(* Schneider Machine Expert - Basic project AND Gate, file version 2.9.0.0 *)
(* ProjectInformations: Name=New project *)

HARDWARE
  Cpu 0: TM221C24R
  EthernetConfiguration: NetworkName=M221, IpAllocationMode=FixedAddress, IpAddress=0.0.0.0, SubnetMask=0.0.0.0
  SerialLineConfiguration: Baud=Baud19200, Parity=ParityEven, DataBits=DataBits8, StopBits=StopBits1, PhysicalMedium=PhysicalMediumRs485, SlaveId=1, Addressing=SlaveAddressing
  MastTask: UsePeriodScanMode=false, PeriodScan=100
  FastTask: Period=255
  CpuBehavior: StartingMode=StartAsPreviousState, AutoSaveRamOnEeprom=true, WatchdogPeriod=250

SYMBOLS  (address, symbol, comment, settings)
  %I0.0     SWITCH_1
  %I0.1     SWITCH_2
  %I0.2     SWITCH_3
  %Q0.0     LED_1

POU New POU
  (* SectionNumber=1 *)

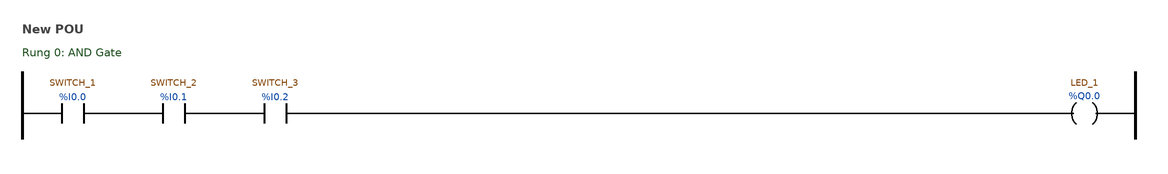

// Rung 0: AND Gate
  LD %I0.0                (* SWITCH_1 *)
  AND %I0.1               (* SWITCH_2 *)
  AND %I0.2               (* SWITCH_3 *)
  ST %Q0.0                (* LED_1 *)
  // as ST:
  //   LED_1 := SWITCH_1 AND SWITCH_2 AND SWITCH_3;
